{attribute 'linkalways'} 
{attribute 'no_explicit_call' := 'This FB is a CLASS and must be accessed using methods or properties'}
{attribute 'enable_dynamic_creation'}
FUNCTION_BLOCK Node_ContainerType_Vector_TcVnVector2_SINT EXTENDS Node
VAR
    out : _GUID;
END_VAR

METHOD PUBLIC  Clone : I_Node
VAR
	pNode : POINTER TO Node_ContainerType_Vector_TcVnVector2_SINT;
END_VAR
pNode := __NEW(Node_ContainerType_Vector_TcVnVector2_SINT);
Clone := pNode^;
END_METHOD

METHOD FB_init : BOOL
VAR_INPUT
	bInitRetains : BOOL; // if TRUE, the retain variables are initialized (warm start / cold start)
	bInCopyCode : BOOL;  // if TRUE, the instance afterwards gets moved into the copy code (online change)
END_VAR
AddOutput('out', out);
END_METHOD

METHOD PROTECTED OnExecute
out.Value := ContainerType_Vector_TcVnVector2_SINT;
END_METHOD

END_FUNCTION_BLOCK

(* stored: Version 1.1.0.1, ProductVersion 3.1.4026.17
   POU Node_ContainerType_Vector_TcVnVector2_SINT: Id {0d433534-3c73-0399-017f-0eb573a2cc05}, SpecialFunc None
   Folder Constructor: Id {b8fe5cf4-fbfd-0f3d-2a24-2557b06436b9}
   Method Clone: Id {9bb46e2c-eb6e-0f60-39bb-23be57a34bb0}
   Method FB_init: Id {f7614ce7-18be-06bf-05ea-8109f586926d}
   Method OnExecute: Id {699b95a3-e070-0323-0f0d-856e92d3cd84} *)
